// TIA Portal V16 export
// export: Created 2021-03-04T22:04:01.9301615Z, ExportSetting WithDefaults, DisplayName Totally Integrated Automation Portal, DisplayVersion V16, DisplayName TIA Portal Version Control Interface, DisplayVersion V16, DisplayName TIA Portal Openness, DisplayVersion V16, DisplayName SINAMICS Startdrive Advanced, DisplayVersion V16, DisplayName SINAMICS Startdrive G130, G150, S120, S150, SINAMICS MV, S210, DisplayVersion V16, DisplayName SINAMICS Startdrive G110M, G120, G120C, G120D, G120P, DisplayVersion V16, DisplayName STEP 7 Professional, DisplayVersion V16, DisplayName STEP 7 Safety, DisplayVersion V16, DisplayName WinCC Professional, DisplayVersion V16
FUNCTION_BLOCK "fbModbusTCPClient"   // FB12, LAD
{ S7_Optimized_Access := 'TRUE' }
VERSION : 0.1
// stored: AutoNumber true, IsIECCheckEnabled false, IsRetainMemResEnabled false, MemoryReserve 100, SetENOAutomatically false, UDAEnableTagReadback false
   VAR_INPUT
      bInRequest { ExternalAccessible := 'False'; ExternalVisible := 'False'; ExternalWritable := 'False'} : Bool;
      bInReset { ExternalVisible := 'False'} : Bool;
      iInSlaveId { ExternalAccessible := 'False'; ExternalVisible := 'False'; ExternalWritable := 'False'} : UInt;
   END_VAR
   VAR_OUTPUT
      bOutError { ExternalAccessible := 'False'; ExternalVisible := 'False'; ExternalWritable := 'False'} : Bool;
      wOutLastErrorCode { ExternalAccessible := 'False'; ExternalVisible := 'False'; ExternalWritable := 'False'} : Word;
   END_VAR
   VAR_IN_OUT
      InOutConnect : TCON_IP_v4;
      InOutReadDiscreteData : Array[*] of "udtModbusValBool";
      InOutWriteCoilData : Array[*] of "udtModbusValBool";
      InOutReadRegisterData : Array[*] of "udtModbusValReal";
      InOutWriteRegisterData : Array[*] of "udtModbusValReal";
   END_VAR
   VAR
      iState { ExternalAccessible := 'False'; ExternalVisible := 'False'; ExternalWritable := 'False'} : Int;
      iNextState { ExternalAccessible := 'False'; ExternalVisible := 'False'; ExternalWritable := 'False'} : Int;
      insModbusClient_TCP { ExternalAccessible := 'False'; ExternalVisible := 'False'; ExternalWritable := 'False'} : MB_CLIENT;
      bTrigReset { ExternalAccessible := 'False'; ExternalVisible := 'False'; ExternalWritable := 'False'} : Bool;
      bTrigReq { ExternalAccessible := 'False'; ExternalVisible := 'False'; ExternalWritable := 'False'} : Bool;
      iNumReadRegisters { ExternalAccessible := 'False'; ExternalVisible := 'False'; ExternalWritable := 'False'} : DInt;
      iNumWriteRegisters { ExternalAccessible := 'False'; ExternalVisible := 'False'; ExternalWritable := 'False'} : DInt;
      iCurrentRegisterReadIndex { ExternalAccessible := 'False'; ExternalVisible := 'False'; ExternalWritable := 'False'} : DInt;
      iCurrentRegisterWriteIndex { ExternalAccessible := 'False'; ExternalVisible := 'False'; ExternalWritable := 'False'} : DInt;
      arrDataWords { ExternalAccessible := 'False'; ExternalVisible := 'False'; ExternalWritable := 'False'} : Array[0..1] of Word;
      iNumReadDiscrete { ExternalAccessible := 'False'; ExternalVisible := 'False'; ExternalWritable := 'False'} : DInt;
      iCurrentDiscreteReadIndex { ExternalAccessible := 'False'; ExternalVisible := 'False'; ExternalWritable := 'False'} : DInt;
      iCurrentCoilWriteIndex { ExternalAccessible := 'False'; ExternalVisible := 'False'; ExternalWritable := 'False'} : DInt;
      iNumWriteCoils { ExternalAccessible := 'False'; ExternalVisible := 'False'; ExternalWritable := 'False'} : DInt;
   END_VAR
   VAR_TEMP
      iMode : USInt;
      iDataAddr : UDInt;
      tempDWord : DWord;
      bConnect : Bool;
      rTemp : Real;
   END_VAR
   VAR CONSTANT
      MODE_READ : USInt := 0;
      MODE_WRITE : USInt := 1;
      IDLE : Int := 0;
      READ_DISC_INIT : Int := 100;
      READ_DISC : Int := 110;
      READ_DISC_NEXT : Int := 120;
      WRITE_COILS_INIT : Int := 200;
      WRITE_COILS : Int := 210;
      WRITE_COILS_NEXT : Int := 220;
      READ_REGS_INIT : Int := 300;
      READ_REGS : Int := 310;
      READ_REGS_PARSE : Int := 320;
      READ_REGS_NEXT : Int := 330;
      WRITE_REGS_INIT : Int := 400;
      WRITE_REGS : Int := 410;
      WRITE_REGS_READBACK_INIT : Int := 420;
      WRITE_REGS_READBACK : Int := 430;
      WRITE_REGS_READBACK_PARSE : Int := 440;
      WRITE_REGS_NEXT : Int := 450;
   END_VAR
   VAR_TEMP   // added for the SCL form of the ladder/FBD networks
      _w1 : Bool;
      _w2 : Bool;
      _w3 : Bool;
      _w4 : Bool;
      _w5 : Bool;
      _w6 : Bool;
      _w7 : Bool;
      _w8 : Bool;
   END_VAR
BEGIN

REGION Network 1: ------------------------------ State Logic ----------------------------------
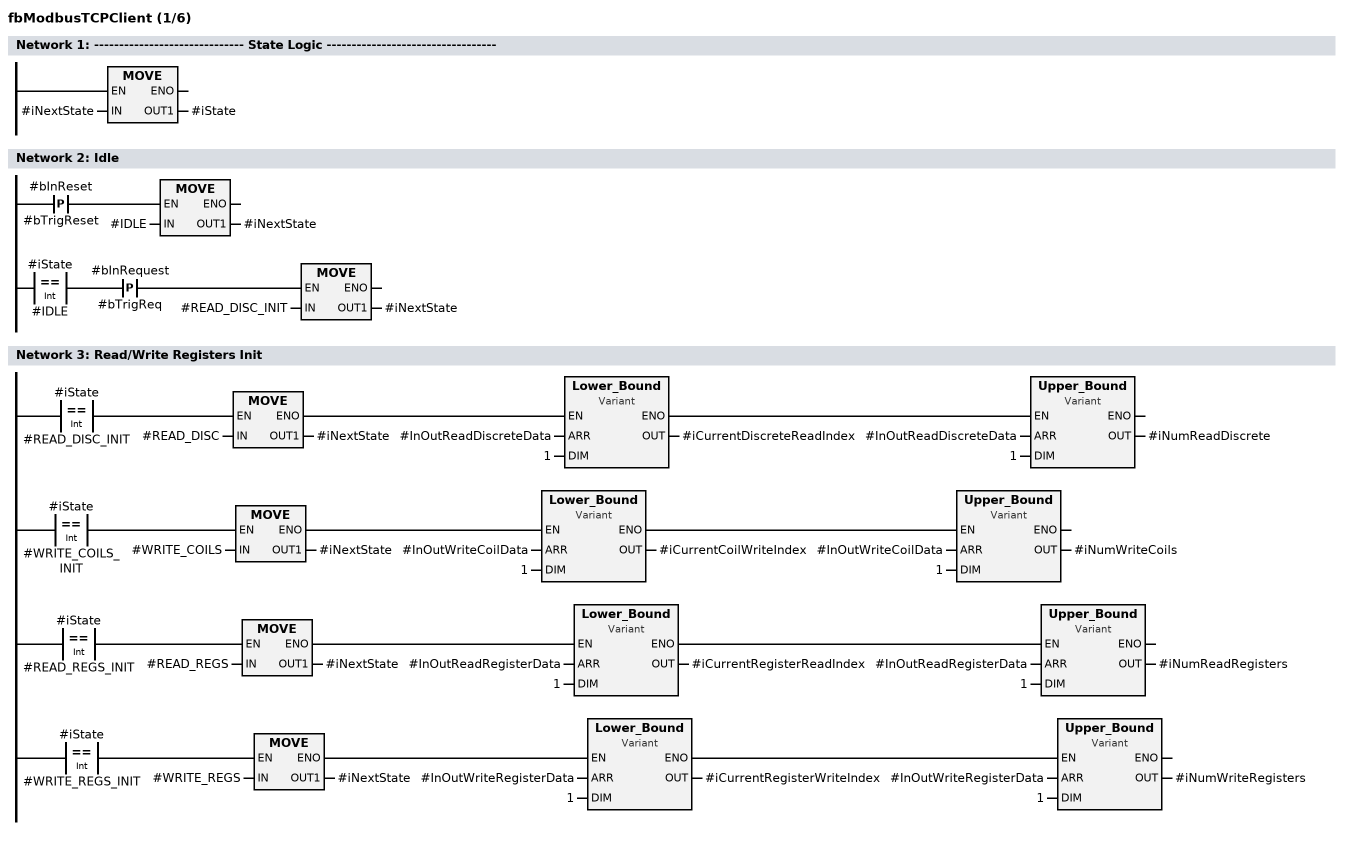
   RUNG wire#powerrail
      Move(in := #iNextState, out1 => #iState)
   END_RUNG
   // the same network as SCL:
   #iState := #iNextState;
END_REGION

REGION Network 2: Idle
   RUNG wire#powerrail
      P_Contact(operand := #bInReset, bit := #bTrigReset)
      Move(in := #IDLE, out1 => #iNextState)
   END_RUNG
   RUNG wire#powerrail
      { S7_Templates := "SrcType := Int" } EQ_Contact(in1 := #iState, in2 := #IDLE)
      P_Contact(operand := #bInRequest, bit := #bTrigReq)
      Move(in := #READ_DISC_INIT, out1 => #iNextState)
   END_RUNG
   // the same network as SCL:
   #_w1 := #bInReset AND NOT #bTrigReset;   // rising edge of #bInReset
   #bTrigReset := #bInReset;
   IF #_w1 THEN #iNextState := #IDLE; END_IF;
   #_w2 := (#iState = #IDLE) AND #bInRequest AND NOT #bTrigReq;   // rising edge of #bInRequest
   #bTrigReq := #bInRequest;
   IF #_w2 THEN #iNextState := #READ_DISC_INIT; END_IF;
END_REGION

REGION Network 3: Read/Write Registers Init
   // no SCL statement known for Lower_Bound, Upper_Bound: written as a call
   // ENO of a box is taken as its EN; it also drops when the box reports an error
   IF #iState = #READ_DISC_INIT THEN
       #iNextState := #READ_DISC;
       Lower_Bound(arr := #InOutReadDiscreteData, dim := 1, out => #iCurrentDiscreteReadIndex);
       Upper_Bound(arr := #InOutReadDiscreteData, dim := 1, out => #iNumReadDiscrete);
   END_IF;
   IF #iState = #WRITE_COILS_INIT THEN
       #iNextState := #WRITE_COILS;
       Lower_Bound(arr := #InOutWriteCoilData, dim := 1, out => #iCurrentCoilWriteIndex);
       Upper_Bound(arr := #InOutWriteCoilData, dim := 1, out => #iNumWriteCoils);
   END_IF;
   IF #iState = #READ_REGS_INIT THEN
       #iNextState := #READ_REGS;
       Lower_Bound(arr := #InOutReadRegisterData, dim := 1, out => #iCurrentRegisterReadIndex);
       Upper_Bound(arr := #InOutReadRegisterData, dim := 1, out => #iNumReadRegisters);
   END_IF;
   IF #iState = #WRITE_REGS_INIT THEN
       #iNextState := #WRITE_REGS;
       Lower_Bound(arr := #InOutWriteRegisterData, dim := 1, out => #iCurrentRegisterWriteIndex);
       Upper_Bound(arr := #InOutWriteRegisterData, dim := 1, out => #iNumWriteRegisters);
   END_IF;
END_REGION

REGION Network 4: Wait for Read/Write to be done
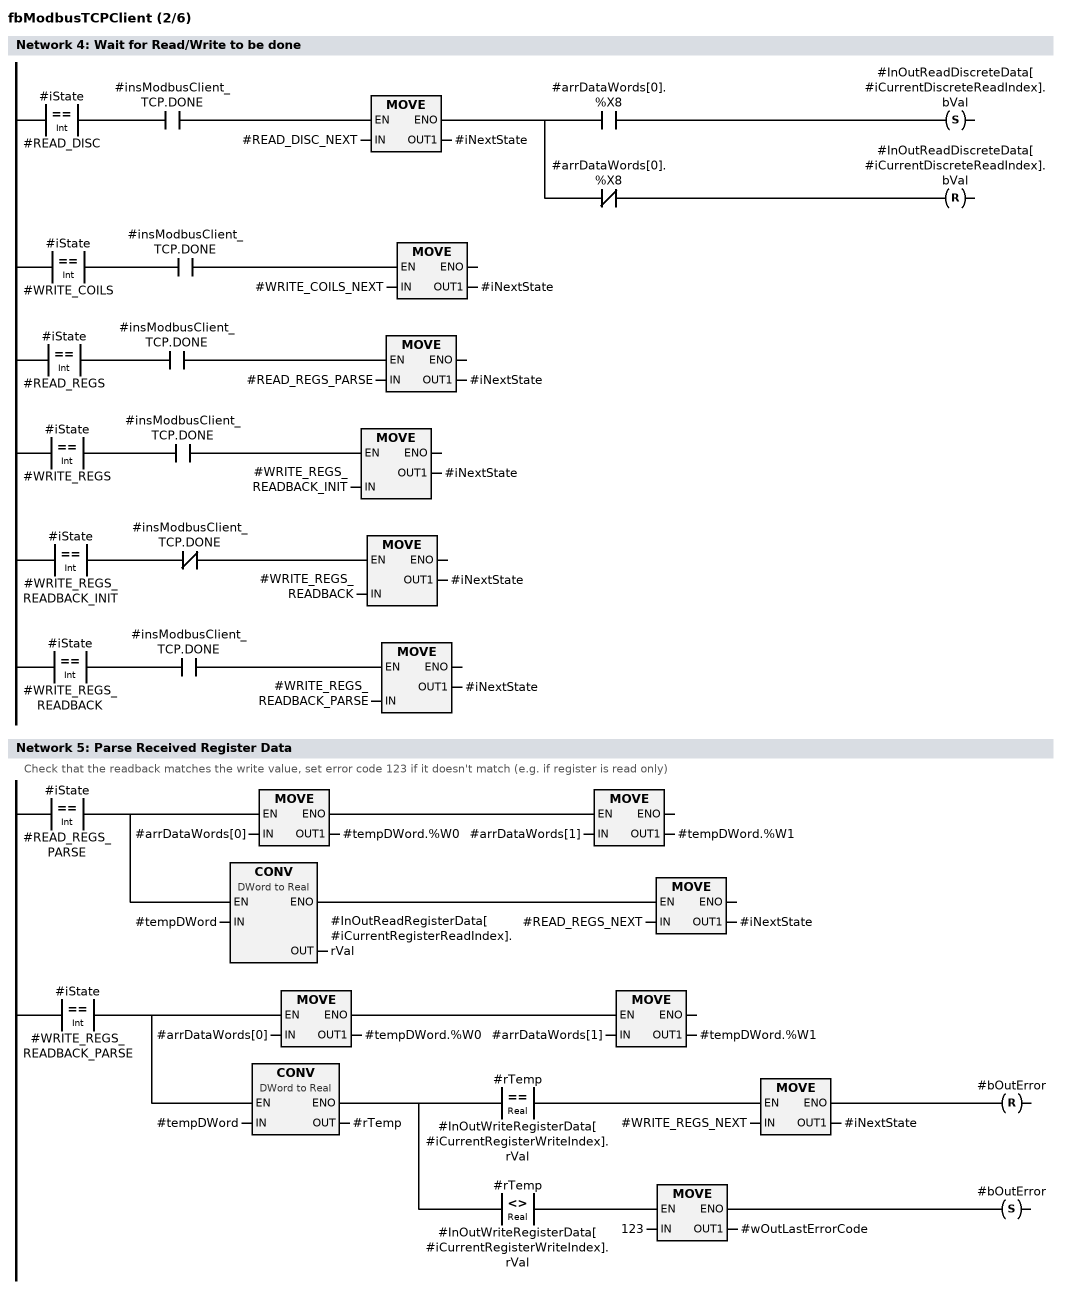
   RUNG wire#powerrail
      { S7_Templates := "SrcType := Int" } EQ_Contact(in1 := #iState, in2 := #READ_DISC)
      Contact( #insModbusClient_TCP.DONE )
      Move(in := #READ_DISC_NEXT, out1 => #iNextState)
      wire#w1
      Contact( #arrDataWords[0].%X8 )
      S_Coil( #InOutReadDiscreteData[#iCurrentDiscreteReadIndex].bVal )
   END_RUNG
   RUNG wire#w1
      I_Contact( #arrDataWords[0].%X8 )
      R_Coil( #InOutReadDiscreteData[#iCurrentDiscreteReadIndex].bVal )
   END_RUNG
   RUNG wire#powerrail
      { S7_Templates := "SrcType := Int" } EQ_Contact(in1 := #iState, in2 := #WRITE_COILS)
      Contact( #insModbusClient_TCP.DONE )
      Move(in := #WRITE_COILS_NEXT, out1 => #iNextState)
   END_RUNG
   RUNG wire#powerrail
      { S7_Templates := "SrcType := Int" } EQ_Contact(in1 := #iState, in2 := #READ_REGS)
      Contact( #insModbusClient_TCP.DONE )
      Move(in := #READ_REGS_PARSE, out1 => #iNextState)
   END_RUNG
   RUNG wire#powerrail
      { S7_Templates := "SrcType := Int" } EQ_Contact(in1 := #iState, in2 := #WRITE_REGS)
      Contact( #insModbusClient_TCP.DONE )
      Move(in := #WRITE_REGS_READBACK_INIT, out1 => #iNextState)
   END_RUNG
   RUNG wire#powerrail
      { S7_Templates := "SrcType := Int" } EQ_Contact(in1 := #iState, in2 := #WRITE_REGS_READBACK_INIT)
      I_Contact( #insModbusClient_TCP.DONE )
      Move(in := #WRITE_REGS_READBACK, out1 => #iNextState)
   END_RUNG
   RUNG wire#powerrail
      { S7_Templates := "SrcType := Int" } EQ_Contact(in1 := #iState, in2 := #WRITE_REGS_READBACK)
      Contact( #insModbusClient_TCP.DONE )
      Move(in := #WRITE_REGS_READBACK_PARSE, out1 => #iNextState)
   END_RUNG
   // the same network as SCL:
   #_w1 := (#iState = #READ_DISC) AND #insModbusClient_TCP.DONE;
   IF #_w1 THEN #iNextState := #READ_DISC_NEXT; END_IF;
   IF #_w1 AND #arrDataWords[0].%X8 THEN
       #InOutReadDiscreteData[#iCurrentDiscreteReadIndex].bVal := TRUE;
   END_IF;
   IF #_w1 AND NOT #arrDataWords[0].%X8 THEN
       #InOutReadDiscreteData[#iCurrentDiscreteReadIndex].bVal := FALSE;
   END_IF;
   IF (#iState = #WRITE_COILS) AND #insModbusClient_TCP.DONE THEN #iNextState := #WRITE_COILS_NEXT; END_IF;
   IF (#iState = #READ_REGS) AND #insModbusClient_TCP.DONE THEN #iNextState := #READ_REGS_PARSE; END_IF;
   IF (#iState = #WRITE_REGS) AND #insModbusClient_TCP.DONE THEN
       #iNextState := #WRITE_REGS_READBACK_INIT;
   END_IF;
   IF (#iState = #WRITE_REGS_READBACK_INIT) AND NOT #insModbusClient_TCP.DONE THEN
       #iNextState := #WRITE_REGS_READBACK;
   END_IF;
   IF (#iState = #WRITE_REGS_READBACK) AND #insModbusClient_TCP.DONE THEN
       #iNextState := #WRITE_REGS_READBACK_PARSE;
   END_IF;
END_REGION

REGION Network 5: Parse Received Register Data
   // Check that the readback matches the write value, set error code 123 if it doesn't match (e.g. if register is read only)
   RUNG wire#powerrail
      { S7_Templates := "SrcType := Int" } EQ_Contact(in1 := #iState, in2 := #READ_REGS_PARSE)
      wire#w1
      Move(in := #arrDataWords[0], out1 => #tempDWord.%W0)
      Move(in := #arrDataWords[1], out1 => #tempDWord.%W1)
   END_RUNG
   RUNG wire#w1
      { S7_Templates := "[SrcType := DWord, DestType := Real]" } Convert(in := #tempDWord, out => #InOutReadRegisterData[#iCurrentRegisterReadIndex].rVal)
      Move(in := #READ_REGS_NEXT, out1 => #iNextState)
   END_RUNG
   RUNG wire#powerrail
      { S7_Templates := "SrcType := Int" } EQ_Contact(in1 := #iState, in2 := #WRITE_REGS_READBACK_PARSE)
      wire#w2
      Move(in := #arrDataWords[0], out1 => #tempDWord.%W0)
      Move(in := #arrDataWords[1], out1 => #tempDWord.%W1)
   END_RUNG
   RUNG wire#w2
      { S7_Templates := "[SrcType := DWord, DestType := Real]" } Convert(in := #tempDWord, out => #rTemp)
      wire#w3
      { S7_Templates := "SrcType := Real" } EQ_Contact(in1 := #rTemp, in2 := #InOutWriteRegisterData[#iCurrentRegisterWriteIndex].rVal)
      Move(in := #WRITE_REGS_NEXT, out1 => #iNextState)
      R_Coil( #bOutError )
   END_RUNG
   RUNG wire#w3
      { S7_Templates := "SrcType := Real" } NE_Contact(in1 := #rTemp, in2 := #InOutWriteRegisterData[#iCurrentRegisterWriteIndex].rVal)
      Move(in := 123, out1 => #wOutLastErrorCode)
      S_Coil( #bOutError )
   END_RUNG
   // the same network as SCL:
   IF #iState = #READ_REGS_PARSE THEN
       #tempDWord.%W0 := #arrDataWords[0];
       #tempDWord.%W1 := #arrDataWords[1];
       #InOutReadRegisterData[#iCurrentRegisterReadIndex].rVal := DWORD_TO_REAL(#tempDWord);
       #iNextState := #READ_REGS_NEXT;
   END_IF;
   #_w1 := #iState = #WRITE_REGS_READBACK_PARSE;
   IF #_w1 THEN
       #tempDWord.%W0 := #arrDataWords[0];
       #tempDWord.%W1 := #arrDataWords[1];
       #rTemp := DWORD_TO_REAL(#tempDWord);
   END_IF;
   IF #_w1 AND (#rTemp = #InOutWriteRegisterData[#iCurrentRegisterWriteIndex].rVal) THEN
       #iNextState := #WRITE_REGS_NEXT;
       #bOutError := FALSE;
   END_IF;
   IF #_w1 AND (#rTemp <> #InOutWriteRegisterData[#iCurrentRegisterWriteIndex].rVal) THEN
       #wOutLastErrorCode := 123;
       #bOutError := TRUE;
   END_IF;
END_REGION

REGION Network 6: Move on to next address
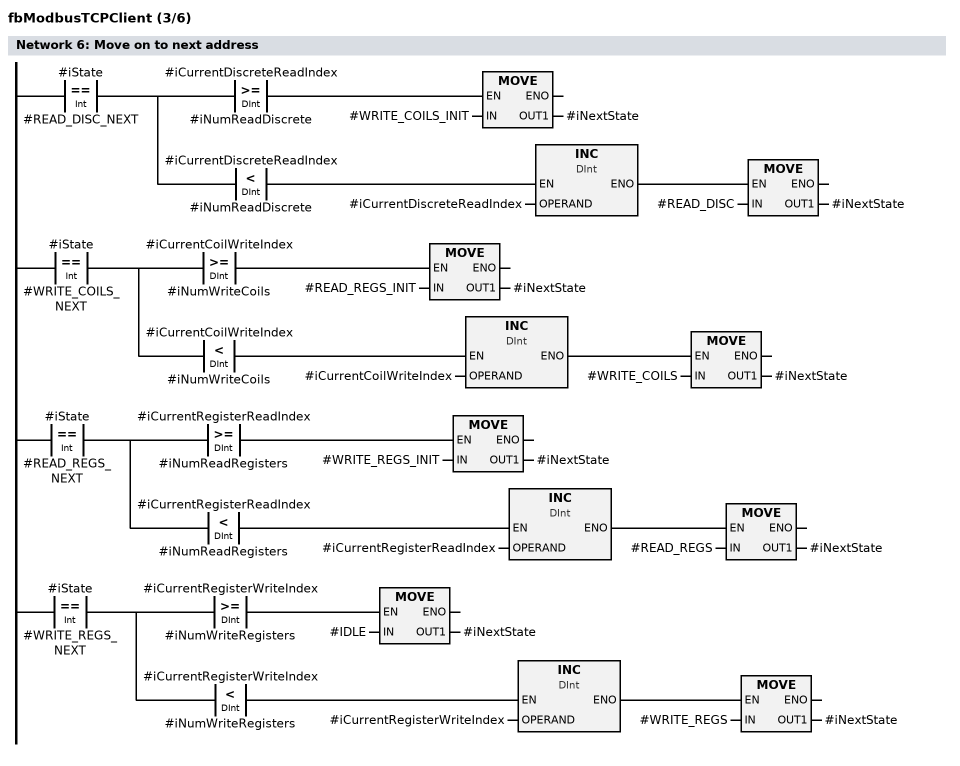
   RUNG wire#powerrail
      { S7_Templates := "SrcType := Int" } EQ_Contact(in1 := #iState, in2 := #READ_DISC_NEXT)
      wire#w1
      { S7_Templates := "SrcType := DInt" } GE_Contact(in1 := #iCurrentDiscreteReadIndex, in2 := #iNumReadDiscrete)
      Move(in := #WRITE_COILS_INIT, out1 => #iNextState)
   END_RUNG
   RUNG wire#w1
      { S7_Templates := "SrcType := DInt" } LT_Contact(in1 := #iCurrentDiscreteReadIndex, in2 := #iNumReadDiscrete)
      { S7_Templates := "DestType := DInt" } Inc( #iCurrentDiscreteReadIndex )
      Move(in := #READ_DISC, out1 => #iNextState)
   END_RUNG
   RUNG wire#powerrail
      { S7_Templates := "SrcType := Int" } EQ_Contact(in1 := #iState, in2 := #WRITE_COILS_NEXT)
      wire#w2
      { S7_Templates := "SrcType := DInt" } GE_Contact(in1 := #iCurrentCoilWriteIndex, in2 := #iNumWriteCoils)
      Move(in := #READ_REGS_INIT, out1 => #iNextState)
   END_RUNG
   RUNG wire#w2
      { S7_Templates := "SrcType := DInt" } LT_Contact(in1 := #iCurrentCoilWriteIndex, in2 := #iNumWriteCoils)
      { S7_Templates := "DestType := DInt" } Inc( #iCurrentCoilWriteIndex )
      Move(in := #WRITE_COILS, out1 => #iNextState)
   END_RUNG
   RUNG wire#powerrail
      { S7_Templates := "SrcType := Int" } EQ_Contact(in1 := #iState, in2 := #READ_REGS_NEXT)
      wire#w3
      { S7_Templates := "SrcType := DInt" } GE_Contact(in1 := #iCurrentRegisterReadIndex, in2 := #iNumReadRegisters)
      Move(in := #WRITE_REGS_INIT, out1 => #iNextState)
   END_RUNG
   RUNG wire#w3
      { S7_Templates := "SrcType := DInt" } LT_Contact(in1 := #iCurrentRegisterReadIndex, in2 := #iNumReadRegisters)
      { S7_Templates := "DestType := DInt" } Inc( #iCurrentRegisterReadIndex )
      Move(in := #READ_REGS, out1 => #iNextState)
   END_RUNG
   RUNG wire#powerrail
      { S7_Templates := "SrcType := Int" } EQ_Contact(in1 := #iState, in2 := #WRITE_REGS_NEXT)
      wire#w4
      { S7_Templates := "SrcType := DInt" } GE_Contact(in1 := #iCurrentRegisterWriteIndex, in2 := #iNumWriteRegisters)
      Move(in := #IDLE, out1 => #iNextState)
   END_RUNG
   RUNG wire#w4
      { S7_Templates := "SrcType := DInt" } LT_Contact(in1 := #iCurrentRegisterWriteIndex, in2 := #iNumWriteRegisters)
      { S7_Templates := "DestType := DInt" } Inc( #iCurrentRegisterWriteIndex )
      Move(in := #WRITE_REGS, out1 => #iNextState)
   END_RUNG
   // the same network as SCL:
   #_w1 := #iState = #READ_DISC_NEXT;
   IF #_w1 AND (#iCurrentDiscreteReadIndex >= #iNumReadDiscrete) THEN
       #iNextState := #WRITE_COILS_INIT;
   END_IF;
   #_w2 := #_w1 AND (#iCurrentDiscreteReadIndex < #iNumReadDiscrete);
   IF #_w2 THEN
       #iCurrentDiscreteReadIndex := #iCurrentDiscreteReadIndex + 1;
       #iNextState := #READ_DISC;
   END_IF;
   #_w3 := #iState = #WRITE_COILS_NEXT;
   IF #_w3 AND (#iCurrentCoilWriteIndex >= #iNumWriteCoils) THEN #iNextState := #READ_REGS_INIT; END_IF;
   #_w4 := #_w3 AND (#iCurrentCoilWriteIndex < #iNumWriteCoils);
   IF #_w4 THEN
       #iCurrentCoilWriteIndex := #iCurrentCoilWriteIndex + 1;
       #iNextState := #WRITE_COILS;
   END_IF;
   #_w5 := #iState = #READ_REGS_NEXT;
   IF #_w5 AND (#iCurrentRegisterReadIndex >= #iNumReadRegisters) THEN
       #iNextState := #WRITE_REGS_INIT;
   END_IF;
   #_w6 := #_w5 AND (#iCurrentRegisterReadIndex < #iNumReadRegisters);
   IF #_w6 THEN
       #iCurrentRegisterReadIndex := #iCurrentRegisterReadIndex + 1;
       #iNextState := #READ_REGS;
   END_IF;
   #_w7 := #iState = #WRITE_REGS_NEXT;
   IF #_w7 AND (#iCurrentRegisterWriteIndex >= #iNumWriteRegisters) THEN #iNextState := #IDLE; END_IF;
   #_w8 := #_w7 AND (#iCurrentRegisterWriteIndex < #iNumWriteRegisters);
   IF #_w8 THEN
       #iCurrentRegisterWriteIndex := #iCurrentRegisterWriteIndex + 1;
       #iNextState := #WRITE_REGS;
   END_IF;
END_REGION

REGION Network 7: ------------------------------ Configure settings and call MB_CLIENT ----------------------------------
END_REGION

REGION Network 8: Set register and data bytes based on array index
   // Assuming that all input address data is formatted with full Modbus address offsets, i.e. coils (00001), discrete inputs (10001), input registers (30001), holding registers (40001)
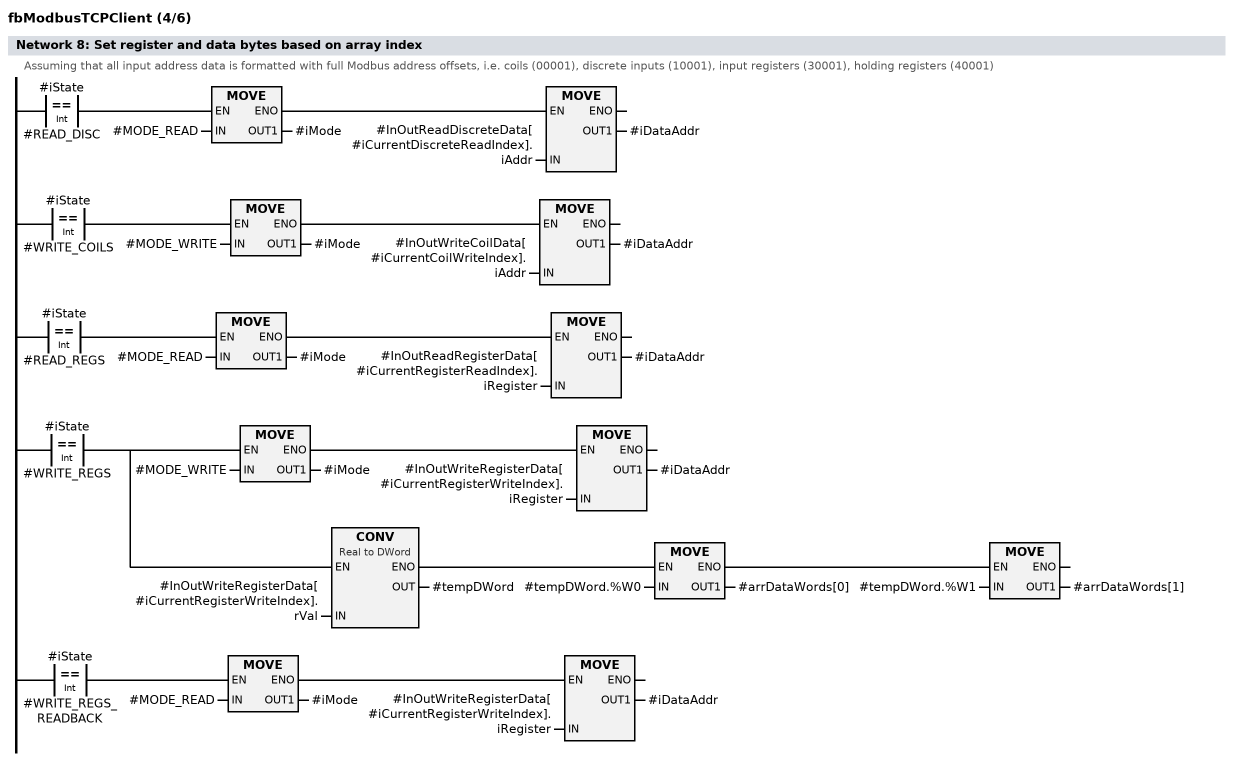
   RUNG wire#powerrail
      { S7_Templates := "SrcType := Int" } EQ_Contact(in1 := #iState, in2 := #READ_DISC)
      Move(in := #MODE_READ, out1 => #iMode)
      Move(in := #InOutReadDiscreteData[#iCurrentDiscreteReadIndex].iAddr, out1 => #iDataAddr)
   END_RUNG
   RUNG wire#powerrail
      { S7_Templates := "SrcType := Int" } EQ_Contact(in1 := #iState, in2 := #WRITE_COILS)
      Move(in := #MODE_WRITE, out1 => #iMode)
      Move(in := #InOutWriteCoilData[#iCurrentCoilWriteIndex].iAddr, out1 => #iDataAddr)
   END_RUNG
   RUNG wire#powerrail
      { S7_Templates := "SrcType := Int" } EQ_Contact(in1 := #iState, in2 := #READ_REGS)
      Move(in := #MODE_READ, out1 => #iMode)
      Move(in := #InOutReadRegisterData[#iCurrentRegisterReadIndex].iRegister, out1 => #iDataAddr)
   END_RUNG
   RUNG wire#powerrail
      { S7_Templates := "SrcType := Int" } EQ_Contact(in1 := #iState, in2 := #WRITE_REGS)
      wire#w1
      Move(in := #MODE_WRITE, out1 => #iMode)
      Move(in := #InOutWriteRegisterData[#iCurrentRegisterWriteIndex].iRegister, out1 => #iDataAddr)
   END_RUNG
   RUNG wire#w1
      { S7_Templates := "[SrcType := Real, DestType := DWord]" } Convert(in := #InOutWriteRegisterData[#iCurrentRegisterWriteIndex].rVal, out => #tempDWord)
      Move(in := #tempDWord.%W0, out1 => #arrDataWords[0])
      Move(in := #tempDWord.%W1, out1 => #arrDataWords[1])
   END_RUNG
   RUNG wire#powerrail
      { S7_Templates := "SrcType := Int" } EQ_Contact(in1 := #iState, in2 := #WRITE_REGS_READBACK)
      Move(in := #MODE_READ, out1 => #iMode)
      Move(in := #InOutWriteRegisterData[#iCurrentRegisterWriteIndex].iRegister, out1 => #iDataAddr)
   END_RUNG
   // the same network as SCL:
   IF #iState = #READ_DISC THEN
       #iMode := #MODE_READ;
       #iDataAddr := #InOutReadDiscreteData[#iCurrentDiscreteReadIndex].iAddr;
   END_IF;
   IF #iState = #WRITE_COILS THEN
       #iMode := #MODE_WRITE;
       #iDataAddr := #InOutWriteCoilData[#iCurrentCoilWriteIndex].iAddr;
   END_IF;
   IF #iState = #READ_REGS THEN
       #iMode := #MODE_READ;
       #iDataAddr := #InOutReadRegisterData[#iCurrentRegisterReadIndex].iRegister;
   END_IF;
   IF #iState = #WRITE_REGS THEN
       #iMode := #MODE_WRITE;
       #iDataAddr := #InOutWriteRegisterData[#iCurrentRegisterWriteIndex].iRegister;
       #tempDWord := REAL_TO_DWORD(#InOutWriteRegisterData[#iCurrentRegisterWriteIndex].rVal);
       #arrDataWords[0] := #tempDWord.%W0;
       #arrDataWords[1] := #tempDWord.%W1;
   END_IF;
   IF #iState = #WRITE_REGS_READBACK THEN
       #iMode := #MODE_READ;
       #iDataAddr := #InOutWriteRegisterData[#iCurrentRegisterWriteIndex].iRegister;
   END_IF;
END_REGION

REGION Network 9: MB_CLIENT block call
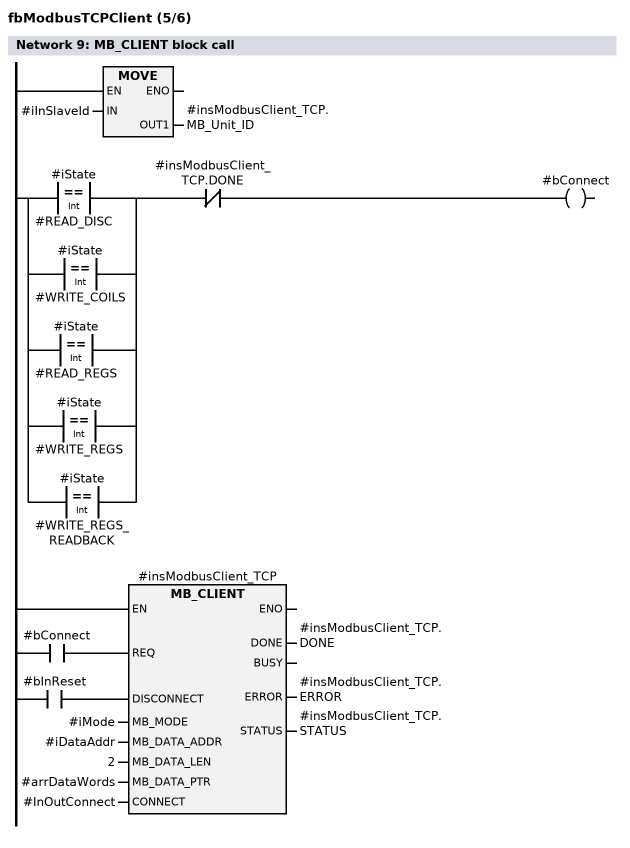
   RUNG wire#powerrail
      Move(in := #iInSlaveId, out1 => #insModbusClient_TCP.MB_Unit_ID)
   END_RUNG
   RUNG wire#powerrail
      { S7_Templates := "SrcType := Int" } EQ_Contact(in1 := #iState, in2 := #READ_DISC)
      wire#w1
      I_Contact( #insModbusClient_TCP.DONE )
      Coil( #bConnect )
   END_RUNG
   RUNG wire#powerrail
      { S7_Templates := "SrcType := Int" } EQ_Contact(in1 := #iState, in2 := #WRITE_COILS)
   END_RUNG wire#w1
   RUNG wire#powerrail
      { S7_Templates := "SrcType := Int" } EQ_Contact(in1 := #iState, in2 := #READ_REGS)
   END_RUNG wire#w1
   RUNG wire#powerrail
      { S7_Templates := "SrcType := Int" } EQ_Contact(in1 := #iState, in2 := #WRITE_REGS)
   END_RUNG wire#w1
   RUNG wire#powerrail
      { S7_Templates := "SrcType := Int" } EQ_Contact(in1 := #iState, in2 := #WRITE_REGS_READBACK)
   END_RUNG wire#w1
   RUNG wire#powerrail
      #insModbusClient_TCP.MB_CLIENT(REQ := wire#w2, DISCONNECT := wire#w3, MB_MODE := #iMode, MB_DATA_ADDR := #iDataAddr, MB_DATA_LEN := 2, MB_DATA_PTR := #arrDataWords, CONNECT := #InOutConnect, DONE => #insModbusClient_TCP.DONE, BUSY =>, ERROR => #insModbusClient_TCP.ERROR, STATUS => #insModbusClient_TCP.STATUS)
   END_RUNG
   RUNG wire#powerrail
      Contact( #bConnect )
   END_RUNG wire#w2
   RUNG wire#powerrail
      Contact( #bInReset )
   END_RUNG wire#w3
   // the same network as SCL:
   #insModbusClient_TCP.MB_Unit_ID := #iInSlaveId;
   #bConnect := ((#iState = #READ_DISC) OR (#iState = #WRITE_COILS) OR (#iState = #READ_REGS) OR (#iState = #WRITE_REGS) OR (#iState = #WRITE_REGS_READBACK)) AND NOT #insModbusClient_TCP.DONE;
   #insModbusClient_TCP(REQ := #bConnect,   // MB_CLIENT
                        DISCONNECT := #bInReset,
                        MB_MODE := #iMode,
                        MB_DATA_ADDR := #iDataAddr,
                        MB_DATA_LEN := 2,
                        MB_DATA_PTR := #arrDataWords,
                        CONNECT := #InOutConnect,
                        DONE => #insModbusClient_TCP.DONE,
                        ERROR => #insModbusClient_TCP.ERROR,
                        STATUS => #insModbusClient_TCP.STATUS);
END_REGION

REGION Network 10: Set error status
   // Ignore error code 16#80A3 (same connection already being used)
   // Go back to idle if stuck waiting for read/write
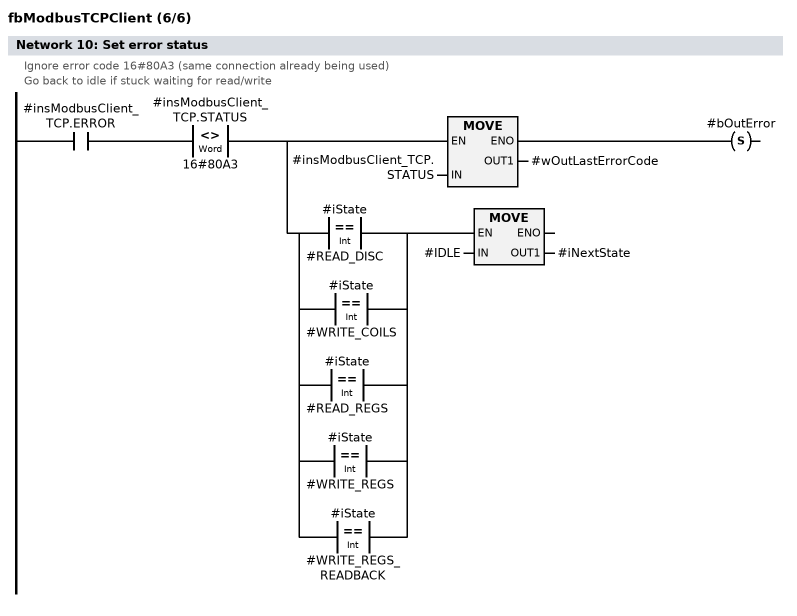
   RUNG wire#powerrail
      Contact( #insModbusClient_TCP.ERROR )
      { S7_Templates := "SrcType := Word" } NE_Contact(in1 := #insModbusClient_TCP.STATUS, in2 := 16#80A3)
      wire#w1
      Move(in := #insModbusClient_TCP.STATUS, out1 => #wOutLastErrorCode)
      S_Coil( #bOutError )
   END_RUNG
   RUNG wire#w1
      { S7_Templates := "SrcType := Int" } EQ_Contact(in1 := #iState, in2 := #READ_DISC)
      wire#w2
      Move(in := #IDLE, out1 => #iNextState)
   END_RUNG
   RUNG wire#w1
      { S7_Templates := "SrcType := Int" } EQ_Contact(in1 := #iState, in2 := #WRITE_COILS)
   END_RUNG wire#w2
   RUNG wire#w1
      { S7_Templates := "SrcType := Int" } EQ_Contact(in1 := #iState, in2 := #READ_REGS)
   END_RUNG wire#w2
   RUNG wire#w1
      { S7_Templates := "SrcType := Int" } EQ_Contact(in1 := #iState, in2 := #WRITE_REGS)
   END_RUNG wire#w2
   RUNG wire#w1
      { S7_Templates := "SrcType := Int" } EQ_Contact(in1 := #iState, in2 := #WRITE_REGS_READBACK)
   END_RUNG wire#w2
   // the same network as SCL:
   #_w1 := #insModbusClient_TCP.ERROR AND (#insModbusClient_TCP.STATUS <> 16#80A3);
   IF #_w1 THEN
       #wOutLastErrorCode := #insModbusClient_TCP.STATUS;
       #bOutError := TRUE;
   END_IF;
   IF #_w1 AND ((#iState = #READ_DISC) OR (#iState = #WRITE_COILS) OR (#iState = #READ_REGS) OR (#iState = #WRITE_REGS) OR (#iState = #WRITE_REGS_READBACK)) THEN
       #iNextState := #IDLE;
   END_IF;
END_REGION
END_FUNCTION_BLOCK
